ABB RobotStudio station: HuiswerkOpdracht.rsstn

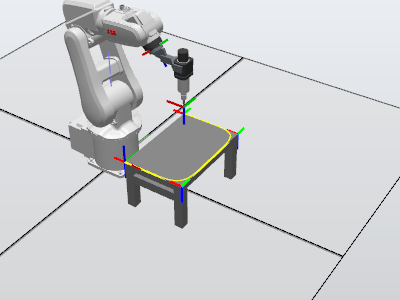
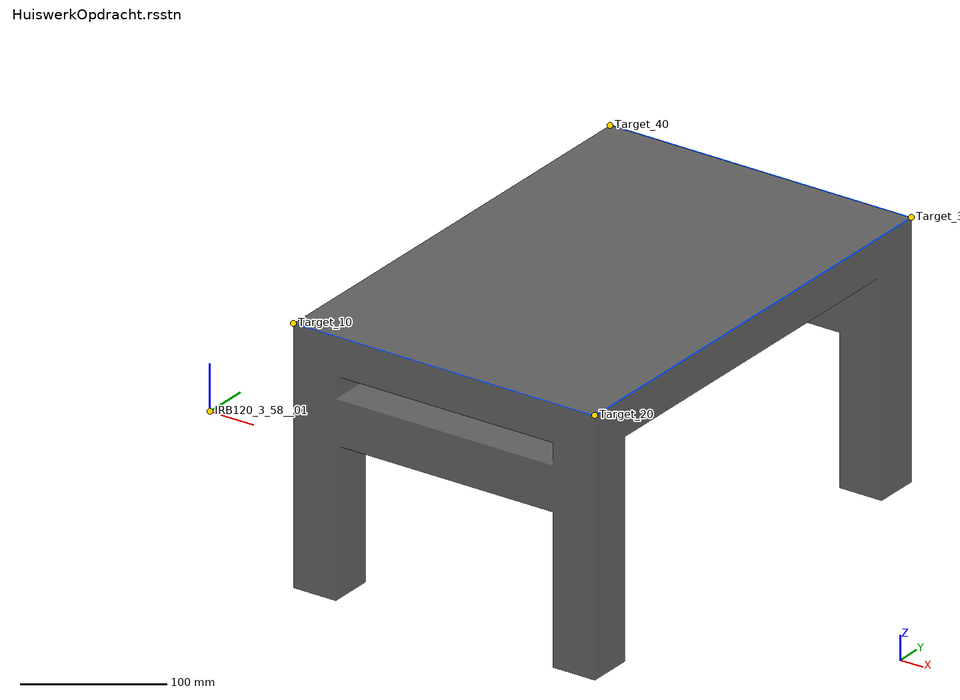
[picture v1: parts stored in the station drawn from their meshes, with robot base, taught points and paths (robot models come from the ABB library and are not in the file)]
Station Station (saved by RobotStudio 23.3.10550.0)
Controller IRB120_3_58
  mechanical unit ROB_1: IRB120_3_58__01, 6 joints, base frame (0, 0, 0) mm
Layout (positions relative to the parent item):
  - IRB120_3_58__01 [mechanism, from %ABB.RobotStudio.Models.IRB120%\IRB120_3_58_G_01.rslib] at (0, 0, 0) mm; joint values [-0.1274, -0.3628, 0.2111, 0.0895, 1.0649, -0.144] (rad or m)
  - Table [part] at (203.21, -191, 0) mm, size 250 x 375 x 200 mm
  - MyTool_2 [mechanism, from Training Objects\myTool.rslib] at (234.9, -24.41, 600.53) mm, rotated rx -180 ry 38 rz 180 deg
Attachment: MyTool_2 is attached to IRB120_3_58__01 / Link6
Attachment: drawing_table is attached to Table
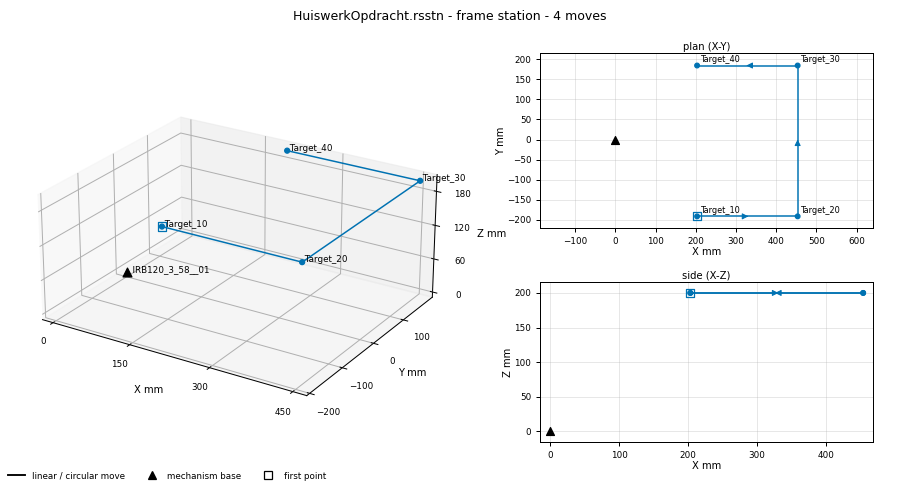
[picture p0: tool path of HuiswerkOpdracht.rsstn in frame station, 4 of 4 moves have a stored position in this frame; points joined in program order, loops and branches not executed]
Targets, tools, work objects and paths stored in the station, written as RAPID:
! task T_ROB1
MODULE CalibData
  PERS tooldata MyTool:=[TRUE,[[31.792631019,0,229.638935148],[0.945518576,0,0.325568154,0]],[1,[0,0,1],[1,0,0,0],0,0,0]];
  TASK PERS wobjdata drawing_table:=[FALSE,TRUE,"",[[-261.354374885,20.903762739,0],[1,0,0,0]],[[464.568,-211.905,200],[1,0,0,0]]];
ENDMODULE

! task T_ROB1
MODULE MainModule
  CONST robtarget Target_10:=[[0.000051301,-0.000031434,-0.000048371],[-0.000000041,0.000000004,1,-0.000000019],[-1,0,-2,0],[9E+09,9E+09,9E+09,9E+09,9E+09,9E+09]];
  CONST robtarget Target_20:=[[250.000075824,0.000012287,-0.000060576],[-0.000000055,-0.000000032,1,-0.000000002],[-1,0,-1,0],[9E+09,9E+09,9E+09,9E+09,9E+09,9E+09]];
  CONST robtarget Target_30:=[[250.000070981,374.999998418,-0.000063071],[-0.000000061,-0.000000008,1,-0.000000014],[0,-1,0,0],[9E+09,9E+09,9E+09,9E+09,9E+09,9E+09]];
  CONST robtarget Target_40:=[[0.000051468,375.000023281,-0.000057615],[-0.00000005,-0.000000036,1,-0.000000013],[0,-1,1,0],[9E+09,9E+09,9E+09,9E+09,9E+09,9E+09]];
  PROC Path_10()
    MoveL Target_10,v1000,z100,MyTool\WObj:=drawing_table;
    MoveL Target_20,v1000,z100,MyTool\WObj:=drawing_table;
    MoveL Target_30,v1000,z100,MyTool\WObj:=drawing_table;
    MoveL Target_40,v1000,z100,MyTool\WObj:=drawing_table;
  ENDPROC
ENDMODULE

